FUNCTION F_NOW_MONOTONIC (* returns current monotonic clock value *)
  (* Standard: 61499-1; Description: Copyright (c) 2024 HR Agrartechnik GmbH This program and the accompanying materials are made available under the terms of the Eclipse Public License 2.0 which is available at https://www.eclipse.org/legal/epl-2.0/ SPDX-License-Identifier: EPL-2.0 return a clear monotonic time monotonic time from a specified point of time (depending on OS and hardware) which has no direct correlation to the current time. (This is only a Wrapper around the ST Function NOW_MONOTONIC) *)
  (* Version 3.0, 2025-04-14, Patrick Aigner, changed package *)
  (* Version 1.0, 2024-10-01, Franz Höpfinger, HR Agrartechnik GmbH *)
  PACKAGE eclipse4diac::utils::timing;
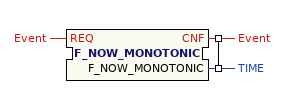
  EVENT_INPUT
    REQ;
  END_EVENT
  EVENT_OUTPUT
    CNF WITH F_NOW_MONOTONIC;
  END_EVENT
  VAR_OUTPUT
    F_NOW_MONOTONIC : TIME;
  END_VAR
  BODY IN ST:
PACKAGE eclipse4diac::utils::timing;

(* returns current monotonic clock value *)
FUNCTION F_NOW_MONOTONIC : TIME
F_NOW_MONOTONIC := NOW_MONOTONIC();
END_FUNCTION
  END_BODY
END_FUNCTION
